(*			
	RAFALOS
	Rafał Osajda		19.09.2025		TC 4024.66
	FB Bazowy dla wszystkich elementów złożonych
*)
FUNCTION_BLOCK FB_BaseComplexElement EXTENDS FB_BaseExecutiveElement IMPLEMENTS ITF_BaseComplexElement, ITF_BaseComplexElement_HMI_Connector
VAR
END_VAR

END_FUNCTION_BLOCK

(* stored: Version 1.1.0.1
   POU FB_BaseComplexElement: Id {1f8518b0-2e03-0c13-2a4a-ffc3b6f9b887}, SpecialFunc None *)
